PROGRAM Tap_proces
VAR
	Step: UINT:=0; 
END_VAR

 CASE Step OF 
	
 	0: 
		IF GVL.Boor_uit AND GVL.Plaat_Gepositioneerd THEN
			Step :=1;
		END_IF

	1:  // Tappen aan zetten
        IF GVL.Tappen_aan THEN
			GVL.Tappen_Start := TRUE;
            Step := 2;
        END_IF
		
    2:  // Tap onderin, Tap gaat terug naar boven
         IF GVL.Tappen_Pos_Bereikt THEN
            GVL.Tappen_Retour := TRUE;
			GVL.Tappen_Start := FALSE;
             Step := 3;
        END_IF

    3:  // Tappen uitzetten
        IF GVL.Tappen_uit THEN
            GVL.Tappen_Retour := FALSE;
            Step := 4;
        END_IF
		
	4:   GVL.Plaat_Gepositioneerd := FALSE;
		 Step:= 1;		

END_CASE

END_PROGRAM

(* stored: Version 1.1.0.1, ProductVersion 3.1.4024.12
   POU Tap_proces: Id {0ac0ace9-0ca8-4fc3-9270-642751849409}, SpecialFunc None *)
